// TIA Portal V16 export
ORGANIZATION_BLOCK "Main"   // OB1, LAD, ProgramCycle
{ S7_Optimized_Access := 'TRUE' }
// stored: AutoNumber false
   VAR_INPUT
      Initial_Call : Bool;
      Remanence : Bool;
   END_VAR
BEGIN

REGION Network 1: Pump control - cyclic LAD call; FirstScan from OB1 Initial_Call
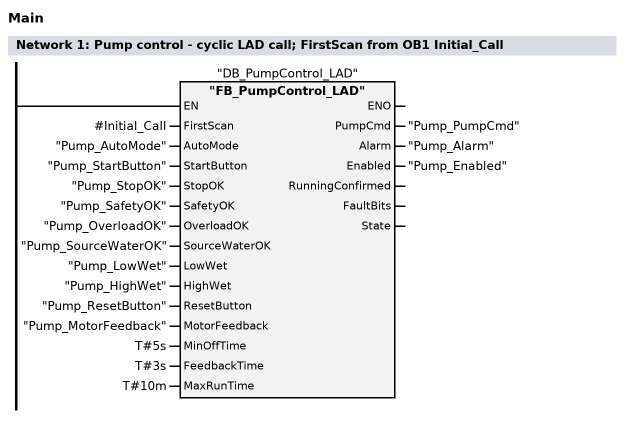
   RUNG wire#powerrail
      "DB_PumpControl_LAD"(FirstScan := #Initial_Call, AutoMode := "Pump_AutoMode", StartButton := "Pump_StartButton", StopOK := "Pump_StopOK", SafetyOK := "Pump_SafetyOK", OverloadOK := "Pump_OverloadOK", SourceWaterOK := "Pump_SourceWaterOK", LowWet := "Pump_LowWet", HighWet := "Pump_HighWet", ResetButton := "Pump_ResetButton", MotorFeedback := "Pump_MotorFeedback", MinOffTime := T#5s, FeedbackTime := T#3s, MaxRunTime := T#10m, PumpCmd => "Pump_PumpCmd", Alarm => "Pump_Alarm", Enabled => "Pump_Enabled", RunningConfirmed =>, FaultBits =>, State =>)
   END_RUNG
   // the same network as SCL:
   "DB_PumpControl_LAD"(FirstScan := #Initial_Call,   // "FB_PumpControl_LAD"
                        AutoMode := "Pump_AutoMode",
                        StartButton := "Pump_StartButton",
                        StopOK := "Pump_StopOK",
                        SafetyOK := "Pump_SafetyOK",
                        OverloadOK := "Pump_OverloadOK",
                        SourceWaterOK := "Pump_SourceWaterOK",
                        LowWet := "Pump_LowWet",
                        HighWet := "Pump_HighWet",
                        ResetButton := "Pump_ResetButton",
                        MotorFeedback := "Pump_MotorFeedback",
                        MinOffTime := T#5s,
                        FeedbackTime := T#3s,
                        MaxRunTime := T#10m,
                        PumpCmd => "Pump_PumpCmd",
                        Alarm => "Pump_Alarm",
                        Enabled => "Pump_Enabled");
END_REGION
END_ORGANIZATION_BLOCK
